TYPE Auto_Test_DB_DUT :
STRUCT
	System: ARRAY[1..5] OF Auto_Test_DUT;
END_STRUCT
END_TYPE

(* stored: Version 1.1.0.1
   DUT Auto_Test_DB_DUT: Id {4a2139bc-7025-4a1d-8cf3-9c1b6954f242} *)
